TYPE UnitAoiHandshaking EXTENDS UnitIndexerSlave :
STRUCT
END_STRUCT
END_TYPE

(* stored: Version 1.1.0.1, ProductVersion 3.1.4020.12
   DUT UnitAoiHandshaking: Id {7d1f4127-d3f1-4cb6-bb57-dae690c6c1dc} *)
